(* Logix 5000 project; controller PeerController vendor 1 type 14 code 196 rev 37.11; software revision 37.00 *)

TASK Hot_Backup_15ms (periodic, rate 15 ms, priority 8, watchdog 500 ms) : Hot_Backup
TASK MainTask (continuous, watchdog 500 ms) : MainProgram

MODULES
   Local : vendor 1 type 14 code 196 (5069 0, rev 37.11)
      Primary : vendor 1 type 14 code 196 (Ethernet 192.168.0.177, rev 37.1, $76aec895$ RPI 10 ms)
      FLEX5000_EIP : 5094-AENTR (Ethernet 192.168.0.179, rev 6.1, StandardDataDriven RPI 200 ms)
         FLEX5000_EIP_SLOT1 : vendor 1 type 7 code 1217 (5094 1, rev 2.1, StandardDataDriven RPI 5 ms)
END_MODULES

TYPE Hot_Backup_Event_Log :
STRUCT
   Event_Name : STRING;
   Value : DINT;
   DateTime : DINT[7];   // Controller Date & Time of the Event
END_STRUCT
END_TYPE

TYPE Hot_Backup_EventLog_Triggers :
STRUCT
   Peer_RunMode : BOOL;
   Peer_ProgramMode : BOOL;
   Peer_ConnectionFailed : BOOL;
   Peer_ConnectionOK : BOOL;
   Peer_Owns_Outputs : BOOL;
   Local_Owns_Outputs : BOOL;
   Manual_SwitchOver_Initiated : BOOL;
   Local_Outputs_Inhibited : BOOL;
   Local_Outputs_Uninhibited : BOOL;
   Peer_Ready : BOOL;
   SwitchoverDelayTimerDone : BOOL;
   Peer_ControllerFault : BOOL;
END_STRUCT
END_TYPE

TYPE Hot_Backup_HMI_Interface :
STRUCT
   ClearEventLog : BOOL;
   Switchover : BOOL;
END_STRUCT
END_TYPE

TYPE Hot_Backup_Interface :
STRUCT
   Sts_ConnectionStatus : CONNECTION_STATUS;   // Produced / Consumed connection status
   Sts_ActionDelay : BOOL;   // Set to "1" when the peer action delay timer is timing.
   Sts_Faulted : BOOL;   // Set to "1" when the peer is faulted
   Sts_OutputsOwned : BOOL;   // Set to "1" when the local controller is the owner of the outputs.
   Sts_OutputInhibitRequest : BOOL;   // Set to "1" when the local controller is manually requesting the peer to inhibit its Outputs
   Fbk_OutputInhibitRequest : BOOL;
END_STRUCT
END_TYPE

ADD_ON_INSTRUCTION Hot_Backup   (* revision 2.0, ExecutePrescan *)
// Compact Logix Hot Backup AOI
VAR_INPUT
   Sts_OutputsInhibited : BOOL; {required}
   Sts_OutputsFaulted : BOOL; {required}
   Cfg_PwrUp_Status : BOOL; {visible}
END_VAR
VAR_OUTPUT
   Cmd_InhibitOutputs : BOOL; {access Read Only, visible}
   Cmd_UninhibitOutputs : BOOL; {access Read Only, visible}
   Sts_PeerReady : BOOL; {access Read Only}
   Sts_Primary : BOOL; {access Read Only, visible}
   Sts_Secondary : BOOL; {access Read Only, visible}
   Sts_PostActionDelay : BOOL; {access Read Only}
END_VAR
VAR_IN_OUT
   PEER_Consumed : Hot_Backup_Interface; {required}
   PEER_Produced : Hot_Backup_Interface; {required}
   HMI_Cmd : Hot_Backup_HMI_Interface; {required}
   HMI_HandShake : Hot_Backup_HMI_Interface; {required}
   HMI_Event_Log : Hot_Backup_Event_Log[10]; {required}   // Contains the 5 most recent event log entries for viewing on the HMI.
END_VAR
VAR
   State : DINT; {access None}
   Int_StartUp_Delay : TIMER := (PRE := 10000); {access None}
   Int_PostAction_Delay : TIMER := (PRE := 60000); {access None}
   State_Processed : BOOL; {access None}
   State_1_Transition : BOOL; {access None}
   State_2_Transition : BOOL; {access None}
   State_3_Transition : BOOL; {access None}
   State_4_Transition : BOOL; {access None}
   ONS : DINT; {access None}
   State_5_Transition : BOOL; {access None}
   Cmd_Inhibit_FromPeer : BOOL; {access None}
   Sts_OutputsOwnerless : BOOL; {access None}
   State_6_Transition : BOOL; {access None}
   Event_Log : Hot_Backup_Event_Log[100];
   Event_Log_Entry : Hot_Backup_Event_Log;
   Event_Log_Index : DINT;
   Event_Log_Name_List : STRING[15] := ([0] := 'Peer in Run Mode', [1] := 'Peer in Program Mode', [2] := 'Peer Connection Failed', [3] := 'Local Outputs Inhibited', [4] := 'Peer Connection OK', [5] := 'Switchover Delay Timer Done', [6] := 'Power Up - First Scan Bit Set', [7] := 'Local Outputs Uninhibited', [8] := 'Peer Owns Outputs', [9] := 'Local Owns Outputs', [10] := 'Manual Switchover Initiated', [11] := 'Peer Controller Major Fault', [12] := 'Peer is Ready');   // Listing of the predefined Event Names
   Event_Log_Triggers : Hot_Backup_EventLog_Triggers; {access None}
   First_Scan : BOOL; {access None}
END_VAR

ROUTINE Logic   (* ladder *)
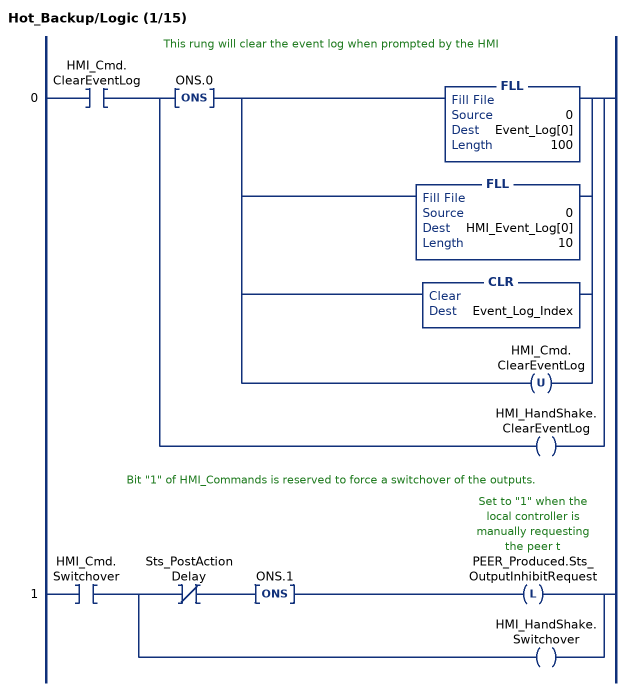
   // This rung will clear the event log when prompted by the HMI
   0: XIC(HMI_Cmd.ClearEventLog)[ONS(ONS.0) [FLL(0,Event_Log[0],100) ,FLL(0,HMI_Event_Log[0],10) ,CLR(Event_Log_Index) ,OTU(HMI_Cmd.ClearEventLog) ] ,OTE(HMI_HandShake.ClearEventLog) ];
   // Bit "1" of HMI_Commands is reserved to force a switchover of the outputs.
   1: XIC(HMI_Cmd.Switchover)[XIO(Sts_PostActionDelay) ONS(ONS.1) OTL(PEER_Produced.Sts_OutputInhibitRequest) ,OTE(HMI_HandShake.Switchover) ];
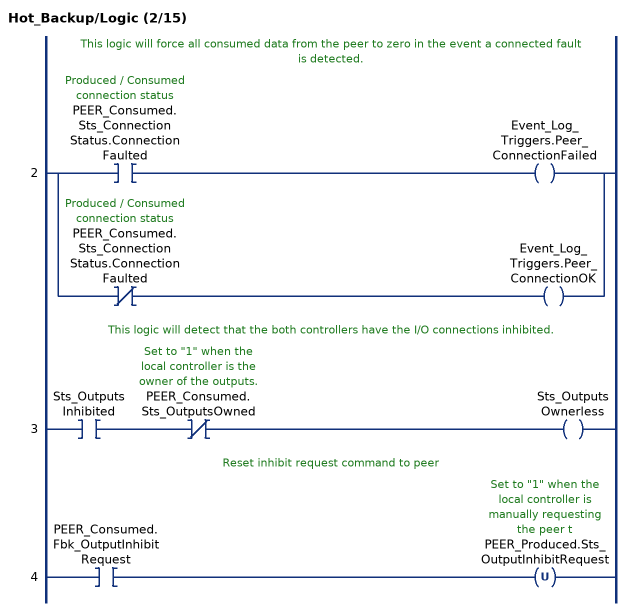
   // This logic will force all consumed data from the peer to zero in the event a connected fault is detected.
   2: [XIC(PEER_Consumed.Sts_ConnectionStatus.ConnectionFaulted) OTE(Event_Log_Triggers.Peer_ConnectionFailed) ,XIO(PEER_Consumed.Sts_ConnectionStatus.ConnectionFaulted) OTE(Event_Log_Triggers.Peer_ConnectionOK) ];
   // This logic will detect that the both controllers have the I/O connections inhibited.
   3: XIC(Sts_OutputsInhibited)XIO(PEER_Consumed.Sts_OutputsOwned)OTE(Sts_OutputsOwnerless);
   // Reset inhibit request command to peer
   4: XIC(PEER_Consumed.Fbk_OutputInhibitRequest)OTU(PEER_Produced.Sts_OutputInhibitRequest);
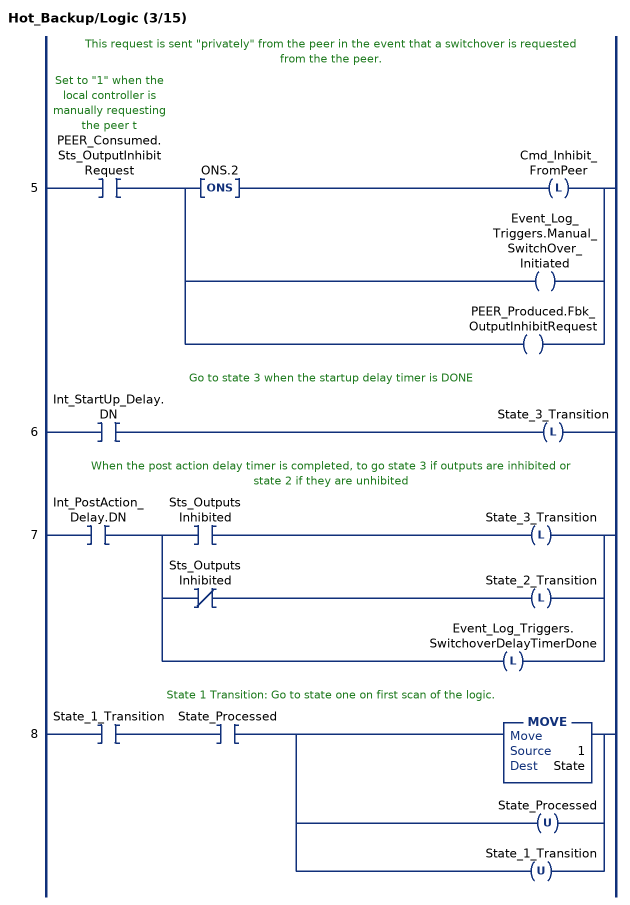
   // This request is sent "privately" from the peer in the event that a switchover is requested from the the peer.
   5: XIC(PEER_Consumed.Sts_OutputInhibitRequest)[ONS(ONS.2) OTL(Cmd_Inhibit_FromPeer) ,OTE(Event_Log_Triggers.Manual_SwitchOver_Initiated) ,OTE(PEER_Produced.Fbk_OutputInhibitRequest) ];
   // Go to state 3 when the startup delay timer is DONE
   6: XIC(Int_StartUp_Delay.DN)OTL(State_3_Transition);
   // When the post action delay timer is completed, to go state 3 if outputs are inhibited or state 2 if they are unhibited
   7: XIC(Int_PostAction_Delay.DN)[XIC(Sts_OutputsInhibited) OTL(State_3_Transition) ,XIO(Sts_OutputsInhibited) OTL(State_2_Transition) ,OTL(Event_Log_Triggers.SwitchoverDelayTimerDone) ];
   // State 1 Transition: Go to state one on first scan of the logic.
   8: XIC(State_1_Transition)XIC(State_Processed)[MOVE(1,State) ,OTU(State_Processed) ,OTU(State_1_Transition) ];
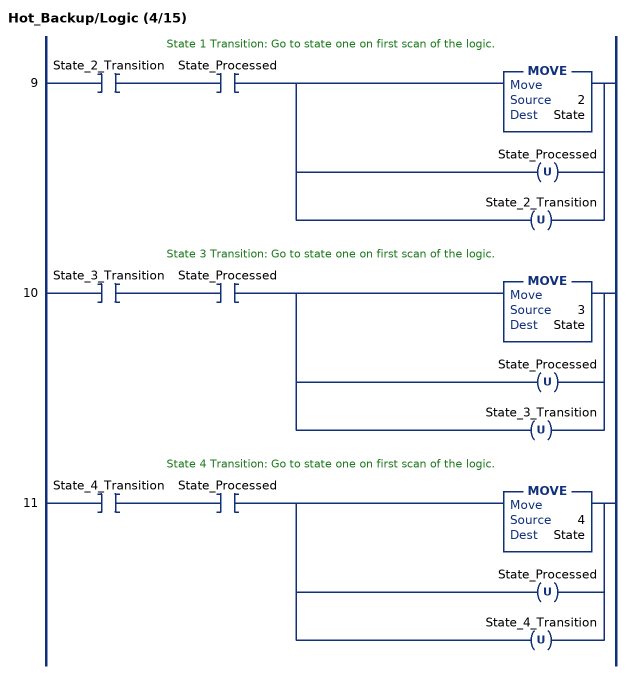
   // State 1 Transition: Go to state one on first scan of the logic.
   9: XIC(State_2_Transition)XIC(State_Processed)[MOVE(2,State) ,OTU(State_Processed) ,OTU(State_2_Transition) ];
   // State 3 Transition: Go to state one on first scan of the logic.
   10: XIC(State_3_Transition)XIC(State_Processed)[MOVE(3,State) ,OTU(State_Processed) ,OTU(State_3_Transition) ];
   // State 4 Transition: Go to state one on first scan of the logic.
   11: XIC(State_4_Transition)XIC(State_Processed)[MOVE(4,State) ,OTU(State_Processed) ,OTU(State_4_Transition) ];
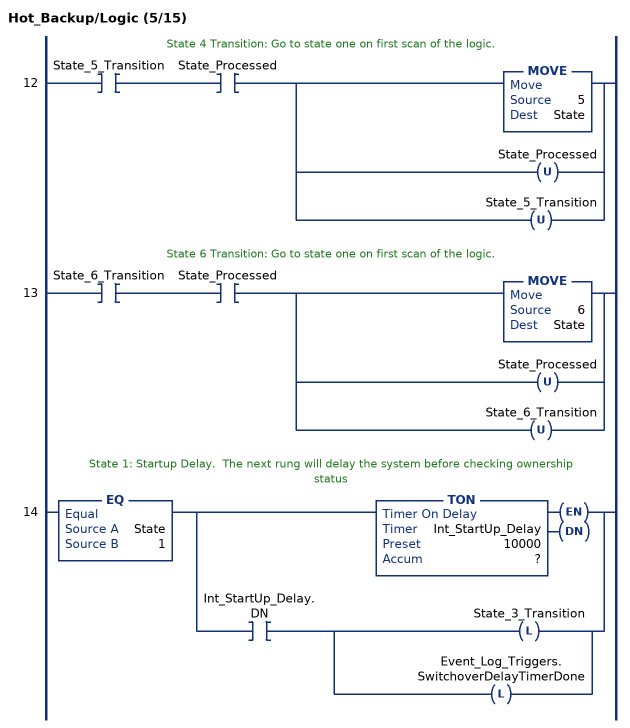
   // State 4 Transition: Go to state one on first scan of the logic.
   12: XIC(State_5_Transition)XIC(State_Processed)[MOVE(5,State) ,OTU(State_Processed) ,OTU(State_5_Transition) ];
   // State 6 Transition: Go to state one on first scan of the logic.
   13: XIC(State_6_Transition)XIC(State_Processed)[MOVE(6,State) ,OTU(State_Processed) ,OTU(State_6_Transition) ];
   // State 1: Startup Delay.  The next rung will delay the system before checking ownership status
   14: EQ(State,1)[TON(Int_StartUp_Delay,?,?) ,XIC(Int_StartUp_Delay.DN) [OTL(State_3_Transition) ,OTL(Event_Log_Triggers.SwitchoverDelayTimerDone) ] ];
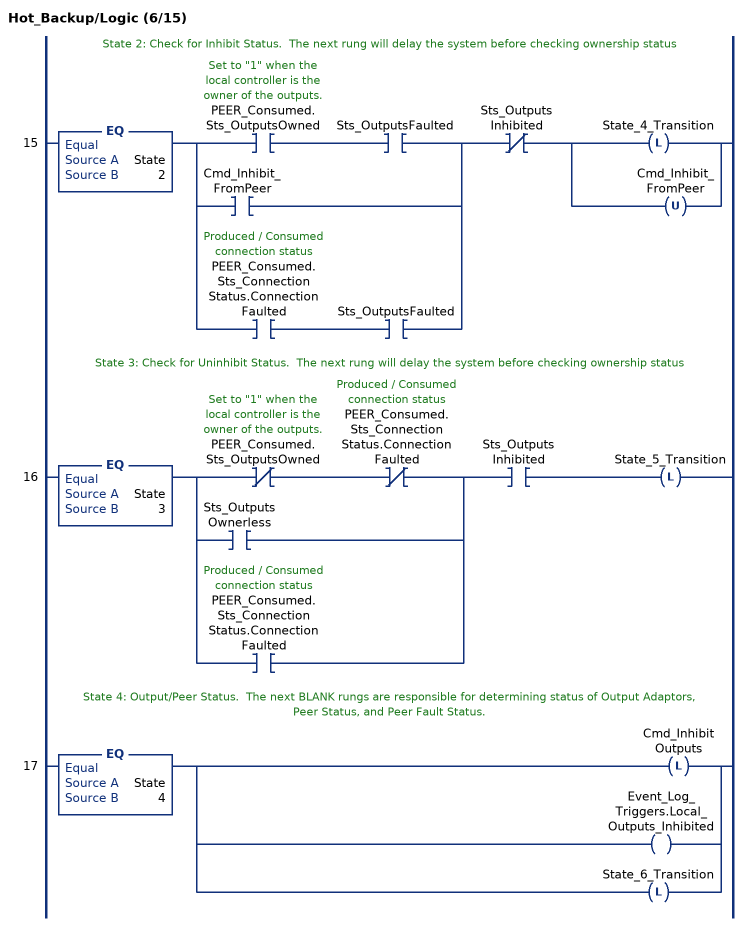
   // State 2: Check for Inhibit Status.  The next rung will delay the system before checking ownership status
   15: EQ(State,2)[XIC(PEER_Consumed.Sts_OutputsOwned) XIC(Sts_OutputsFaulted) ,XIC(Cmd_Inhibit_FromPeer) ,XIC(PEER_Consumed.Sts_ConnectionStatus.ConnectionFaulted) XIC(Sts_OutputsFaulted) ]XIO(Sts_OutputsInhibited)[OTL(State_4_Transition) ,OTU(Cmd_Inhibit_FromPeer) ];
   // State 3: Check for Uninhibit Status.  The next rung will delay the system before checking ownership status
   16: EQ(State,3)[XIO(PEER_Consumed.Sts_OutputsOwned) XIO(PEER_Consumed.Sts_ConnectionStatus.ConnectionFaulted) ,XIC(Sts_OutputsOwnerless) ,XIC(PEER_Consumed.Sts_ConnectionStatus.ConnectionFaulted) ]XIC(Sts_OutputsInhibited)OTL(State_5_Transition);
   // State 4: Output/Peer Status.  The next BLANK rungs are responsible for determining status of Output Adaptors, Peer Status, and Peer Fault Status.
   17: EQ(State,4)[OTL(Cmd_InhibitOutputs) ,OTE(Event_Log_Triggers.Local_Outputs_Inhibited) ,OTL(State_6_Transition) ];
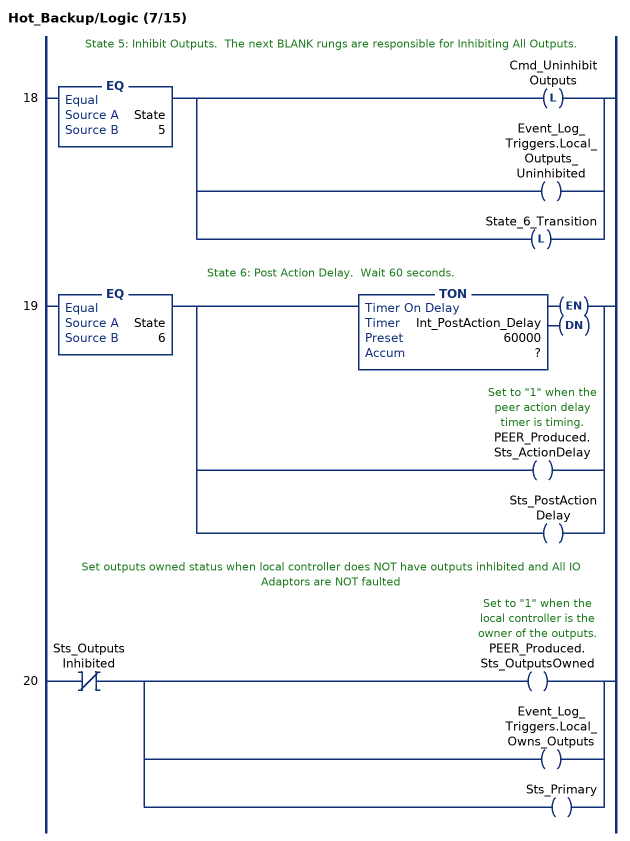
   // State 5: Inhibit Outputs.  The next BLANK rungs are responsible for Inhibiting All Outputs.
   18: EQ(State,5)[OTL(Cmd_UninhibitOutputs) ,OTE(Event_Log_Triggers.Local_Outputs_Uninhibited) ,OTL(State_6_Transition) ];
   // State 6: Post Action Delay.  Wait 60 seconds.
   19: EQ(State,6)[TON(Int_PostAction_Delay,?,?) ,OTE(PEER_Produced.Sts_ActionDelay) ,OTE(Sts_PostActionDelay) ];
   // Set outputs owned status when local controller does NOT have outputs inhibited and All IO Adaptors are NOT faulted
   20: XIO(Sts_OutputsInhibited)[OTE(PEER_Produced.Sts_OutputsOwned) ,OTE(Event_Log_Triggers.Local_Owns_Outputs) ,OTE(Sts_Primary) ];
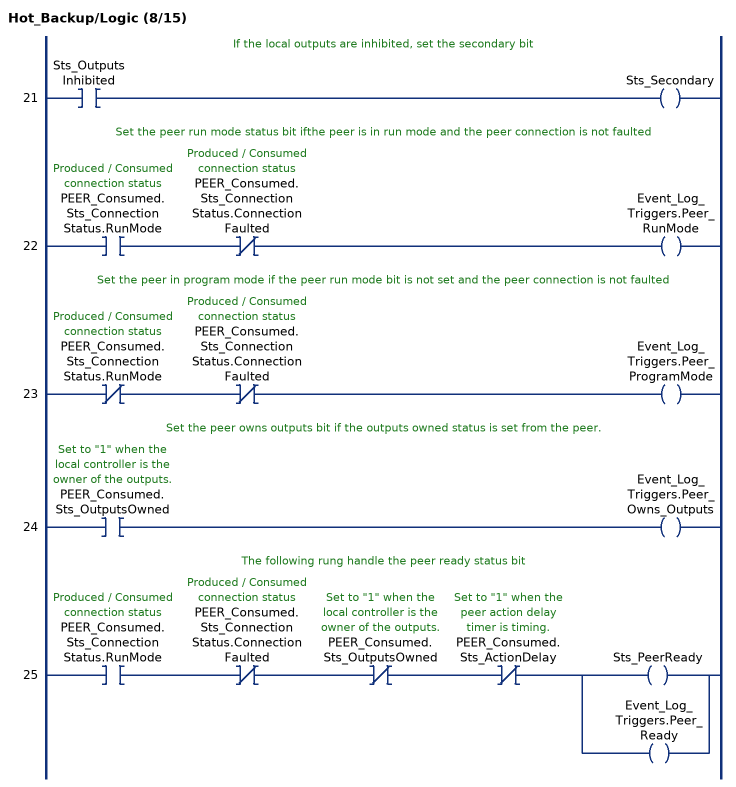
   // If the local outputs are inhibited, set the secondary bit
   21: XIC(Sts_OutputsInhibited)OTE(Sts_Secondary);
   // Set the peer run mode status bit ifthe peer is in run mode and the peer connection is not faulted
   22: XIC(PEER_Consumed.Sts_ConnectionStatus.RunMode)XIO(PEER_Consumed.Sts_ConnectionStatus.ConnectionFaulted)OTE(Event_Log_Triggers.Peer_RunMode);
   // Set the peer in program mode if the peer run mode bit is not set and the peer connection is not faulted
   23: XIO(PEER_Consumed.Sts_ConnectionStatus.RunMode)XIO(PEER_Consumed.Sts_ConnectionStatus.ConnectionFaulted)OTE(Event_Log_Triggers.Peer_ProgramMode);
   // Set the peer owns outputs bit if the outputs owned status is set from the peer.
   24: XIC(PEER_Consumed.Sts_OutputsOwned)OTE(Event_Log_Triggers.Peer_Owns_Outputs);
   // The following rung handle the peer ready status bit
   25: XIC(PEER_Consumed.Sts_ConnectionStatus.RunMode)XIO(PEER_Consumed.Sts_ConnectionStatus.ConnectionFaulted)XIO(PEER_Consumed.Sts_OutputsOwned)XIO(PEER_Consumed.Sts_ActionDelay)[OTE(Sts_PeerReady) ,OTE(Event_Log_Triggers.Peer_Ready) ];
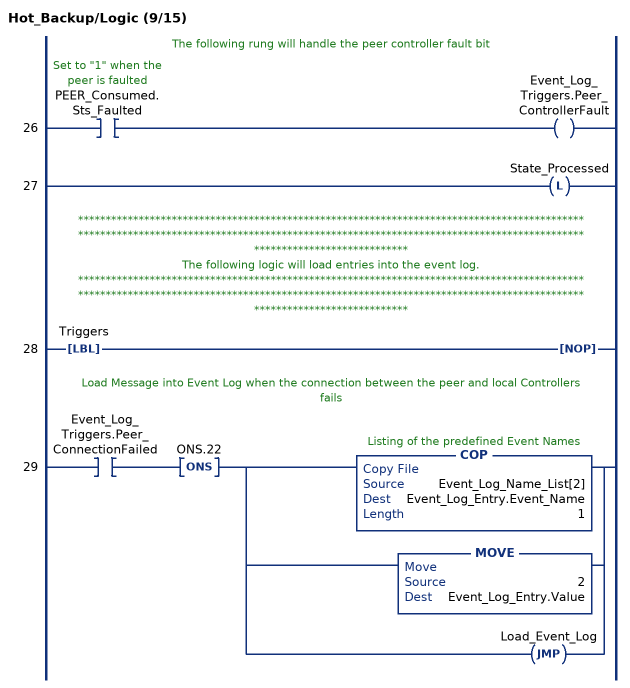
   // The following rung will handle the peer controller fault bit
   26: XIC(PEER_Consumed.Sts_Faulted)OTE(Event_Log_Triggers.Peer_ControllerFault);
   27: OTL(State_Processed);
   // ********************************************************************************************************************************************************************************************************************
   // The following logic will load entries into the event log.
   // ********************************************************************************************************************************************************************************************************************
   28: LBL(Triggers)NOP();
   // Load Message into Event Log when the connection between the peer and local Controllers fails
   29: XIC(Event_Log_Triggers.Peer_ConnectionFailed)ONS(ONS.22)[COP(Event_Log_Name_List[2],Event_Log_Entry.Event_Name,1) ,MOVE(2,Event_Log_Entry.Value) ,JMP(Load_Event_Log) ];
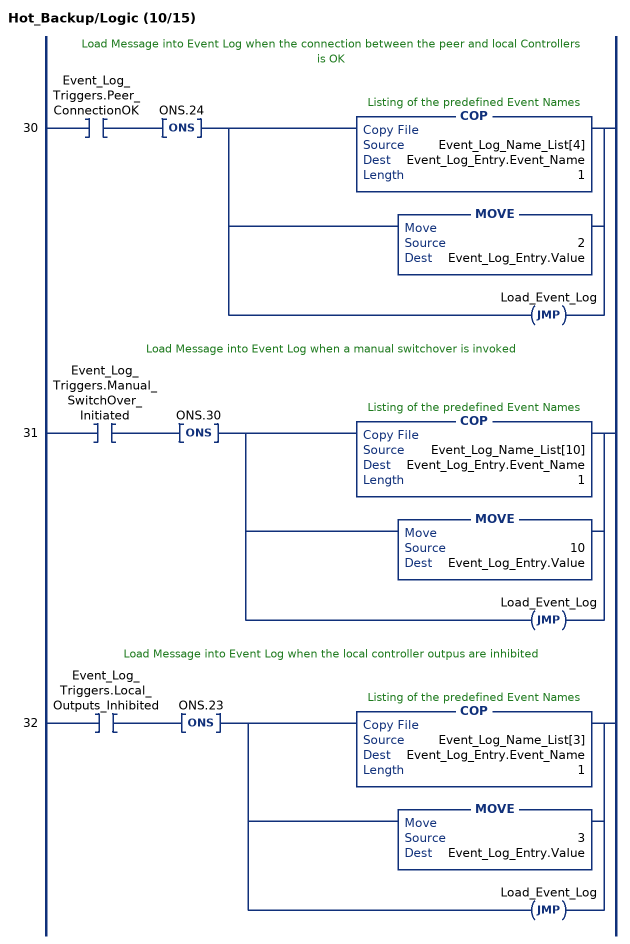
   // Load Message into Event Log when the connection between the peer and local Controllers is OK
   30: XIC(Event_Log_Triggers.Peer_ConnectionOK)ONS(ONS.24)[COP(Event_Log_Name_List[4],Event_Log_Entry.Event_Name,1) ,MOVE(2,Event_Log_Entry.Value) ,JMP(Load_Event_Log) ];
   // Load Message into Event Log when a manual switchover is invoked
   31: XIC(Event_Log_Triggers.Manual_SwitchOver_Initiated)ONS(ONS.30)[COP(Event_Log_Name_List[10],Event_Log_Entry.Event_Name,1) ,MOVE(10,Event_Log_Entry.Value) ,JMP(Load_Event_Log) ];
   // Load Message into Event Log when the local controller outpus are inhibited
   32: XIC(Event_Log_Triggers.Local_Outputs_Inhibited)ONS(ONS.23)[COP(Event_Log_Name_List[3],Event_Log_Entry.Event_Name,1) ,MOVE(3,Event_Log_Entry.Value) ,JMP(Load_Event_Log) ];
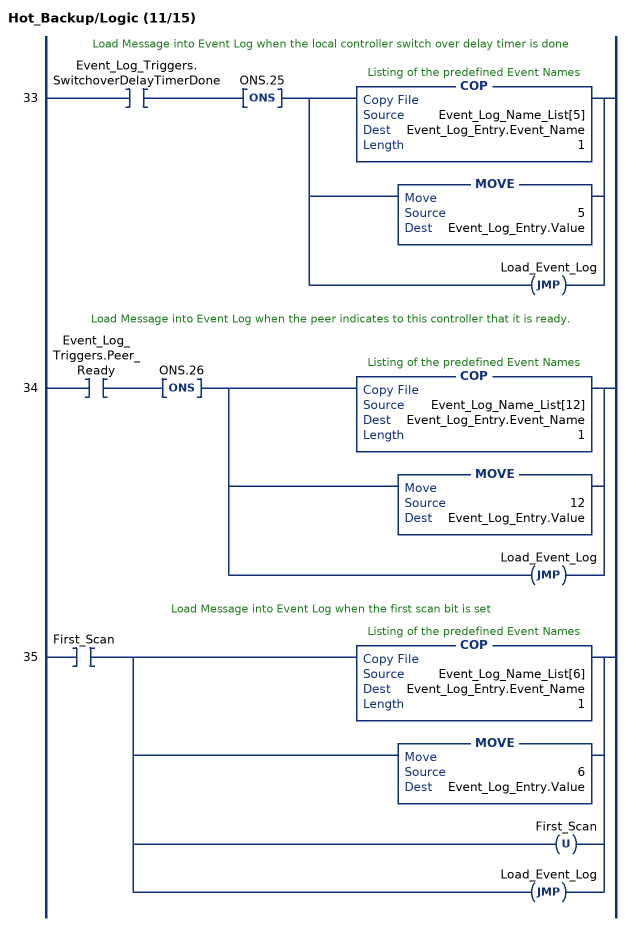
   // Load Message into Event Log when the local controller switch over delay timer is done
   33: XIC(Event_Log_Triggers.SwitchoverDelayTimerDone)ONS(ONS.25)[COP(Event_Log_Name_List[5],Event_Log_Entry.Event_Name,1) ,MOVE(5,Event_Log_Entry.Value) ,JMP(Load_Event_Log) ];
   // Load Message into Event Log when the peer indicates to this controller that it is ready.
   34: XIC(Event_Log_Triggers.Peer_Ready)ONS(ONS.26)[COP(Event_Log_Name_List[12],Event_Log_Entry.Event_Name,1) ,MOVE(12,Event_Log_Entry.Value) ,JMP(Load_Event_Log) ];
   // Load Message into Event Log when the first scan bit is set
   35: XIC(First_Scan)[COP(Event_Log_Name_List[6],Event_Log_Entry.Event_Name,1) ,MOVE(6,Event_Log_Entry.Value) ,OTU(First_Scan) ,JMP(Load_Event_Log) ];
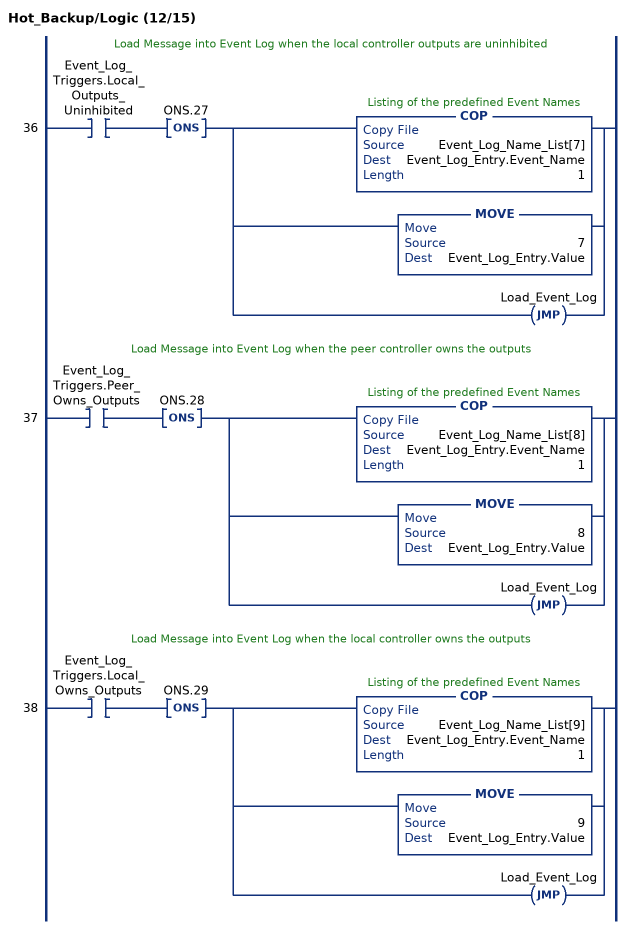
   // Load Message into Event Log when the local controller outputs are uninhibited
   36: XIC(Event_Log_Triggers.Local_Outputs_Uninhibited)ONS(ONS.27)[COP(Event_Log_Name_List[7],Event_Log_Entry.Event_Name,1) ,MOVE(7,Event_Log_Entry.Value) ,JMP(Load_Event_Log) ];
   // Load Message into Event Log when the peer controller owns the outputs
   37: XIC(Event_Log_Triggers.Peer_Owns_Outputs)ONS(ONS.28)[COP(Event_Log_Name_List[8],Event_Log_Entry.Event_Name,1) ,MOVE(8,Event_Log_Entry.Value) ,JMP(Load_Event_Log) ];
   // Load Message into Event Log when the local controller owns the outputs
   38: XIC(Event_Log_Triggers.Local_Owns_Outputs)ONS(ONS.29)[COP(Event_Log_Name_List[9],Event_Log_Entry.Event_Name,1) ,MOVE(9,Event_Log_Entry.Value) ,JMP(Load_Event_Log) ];
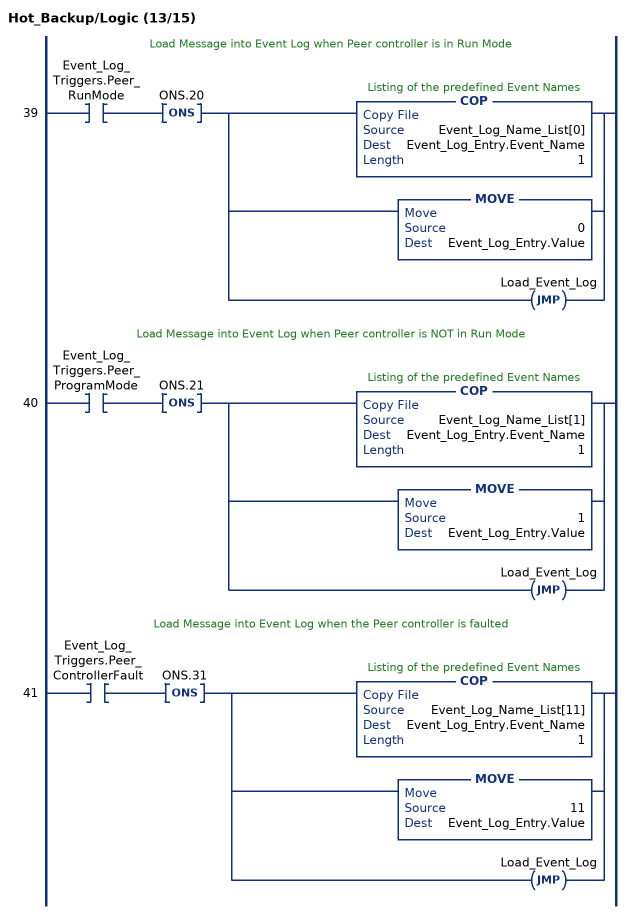
   // Load Message into Event Log when Peer controller is in Run Mode
   39: XIC(Event_Log_Triggers.Peer_RunMode)ONS(ONS.20)[COP(Event_Log_Name_List[0],Event_Log_Entry.Event_Name,1) ,MOVE(0,Event_Log_Entry.Value) ,JMP(Load_Event_Log) ];
   // Load Message into Event Log when Peer controller is NOT in Run Mode
   40: XIC(Event_Log_Triggers.Peer_ProgramMode)ONS(ONS.21)[COP(Event_Log_Name_List[1],Event_Log_Entry.Event_Name,1) ,MOVE(1,Event_Log_Entry.Value) ,JMP(Load_Event_Log) ];
   // Load Message into Event Log when the Peer controller is faulted
   41: XIC(Event_Log_Triggers.Peer_ControllerFault)ONS(ONS.31)[COP(Event_Log_Name_List[11],Event_Log_Entry.Event_Name,1) ,MOVE(11,Event_Log_Entry.Value) ,JMP(Load_Event_Log) ];
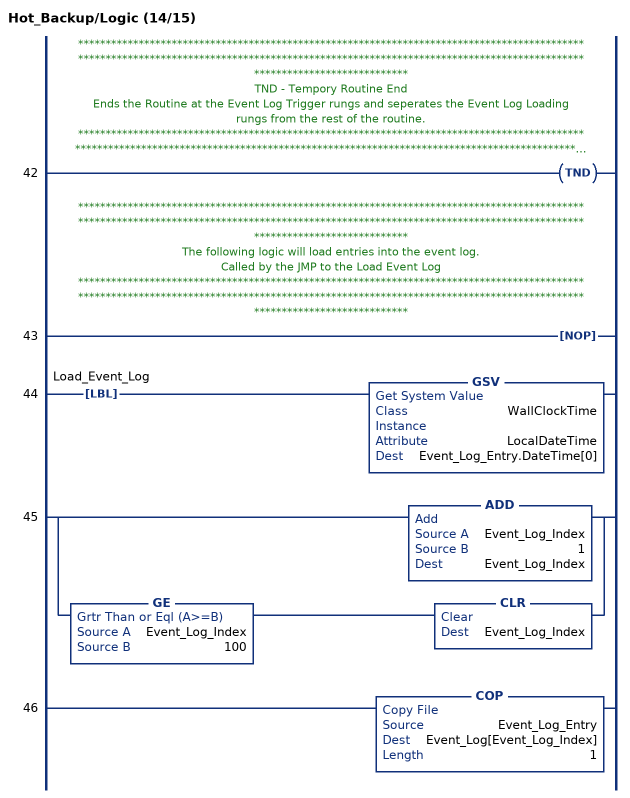
   // ********************************************************************************************************************************************************************************************************************
   // TND - Tempory Routine End
   // Ends the Routine at the Event Log Trigger rungs and seperates the Event Log Loading rungs from the rest of the routine.
   // ********************************************************************************************************************************************************************************************************************
   42: TND();
   // ********************************************************************************************************************************************************************************************************************
   // The following logic will load entries into the event log.
   // Called by the JMP to the Load Event Log
   // ********************************************************************************************************************************************************************************************************************
   43: NOP();
   44: LBL(Load_Event_Log)GSV(WallClockTime,,LocalDateTime,Event_Log_Entry.DateTime[0]);
   45: [ADD(Event_Log_Index,1,Event_Log_Index) ,GE(Event_Log_Index,100) CLR(Event_Log_Index) ];
   46: COP(Event_Log_Entry,Event_Log[Event_Log_Index],1);
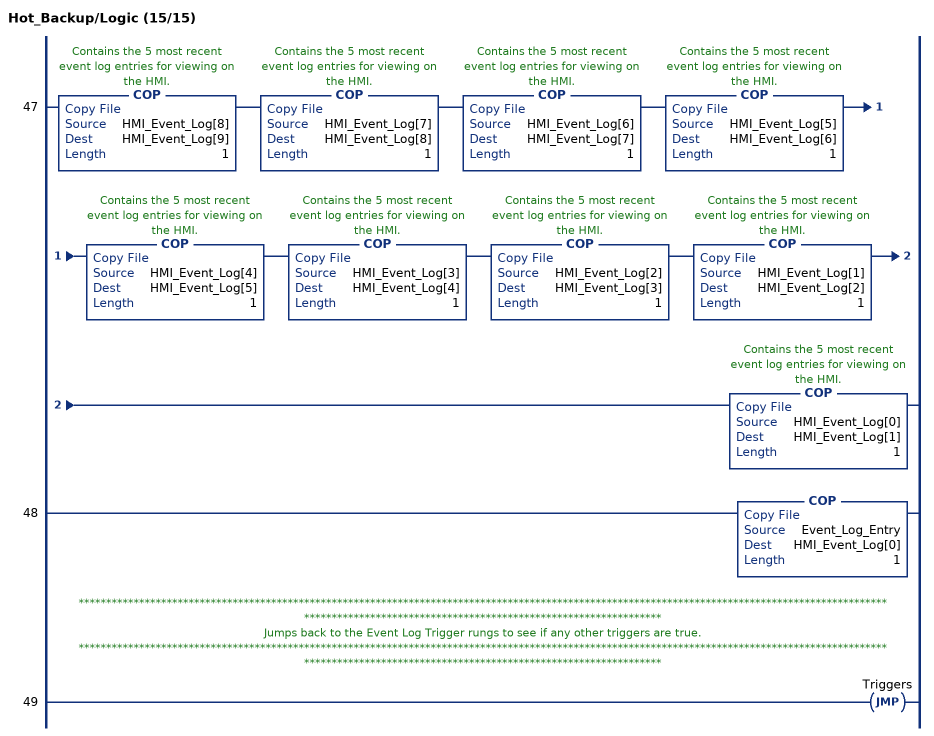
   47: COP(HMI_Event_Log[8],HMI_Event_Log[9],1)COP(HMI_Event_Log[7],HMI_Event_Log[8],1)COP(HMI_Event_Log[6],HMI_Event_Log[7],1)COP(HMI_Event_Log[5],HMI_Event_Log[6],1)COP(HMI_Event_Log[4],HMI_Event_Log[5],1)COP(HMI_Event_Log[3],HMI_Event_Log[4],1)COP(HMI_Event_Log[2],HMI_Event_Log[3],1)COP(HMI_Event_Log[1],HMI_Event_Log[2],1)COP(HMI_Event_Log[0],HMI_Event_Log[1],1);
   48: COP(Event_Log_Entry,HMI_Event_Log[0],1);
   // ********************************************************************************************************************************************************************************************************************
   // Jumps back to the Event Log Trigger rungs to see if any other triggers are true.
   // ********************************************************************************************************************************************************************************************************************
   49: JMP(Triggers);
END_ROUTINE

ROUTINE Prescan   (* ladder *)
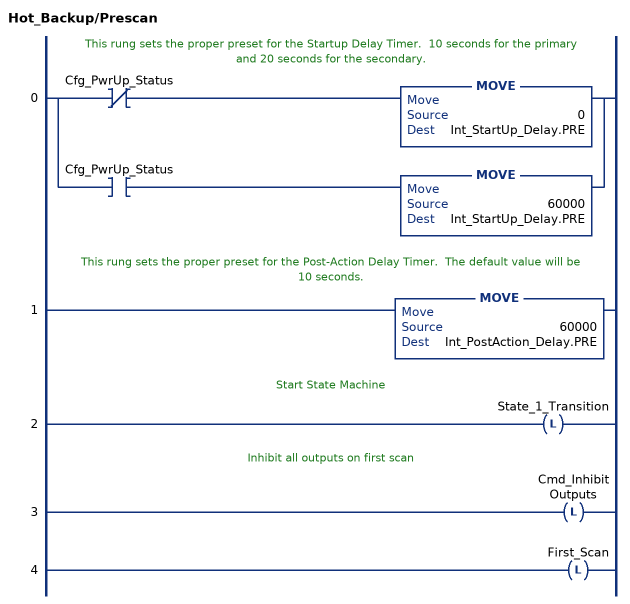
   // This rung sets the proper preset for the Startup Delay Timer.  10 seconds for the primary and 20 seconds for the secondary.
   0: [XIO(Cfg_PwrUp_Status) MOVE(0,Int_StartUp_Delay.PRE) ,XIC(Cfg_PwrUp_Status) MOVE(60000,Int_StartUp_Delay.PRE) ];
   // This rung sets the proper preset for the Post-Action Delay Timer.  The default value will be 10 seconds.
   1: MOVE(60000,Int_PostAction_Delay.PRE);
   // Start State Machine
   2: OTL(State_1_Transition);
   // Inhibit all outputs on first scan
   3: OTL(Cmd_InhibitOutputs);
   4: OTL(First_Scan);
END_ROUTINE
END_ADD_ON_INSTRUCTION

VAR_GLOBAL   (* controller tags *)
   Array : DINT[10];
   DINT : DINT;
   HMI_Cmd : Hot_Backup_HMI_Interface;
   HMI_Event_Log : Hot_Backup_Event_Log[10];
   HMI_Handshake : Hot_Backup_HMI_Interface;
   Manual_Switchover_PB : BOOL;
   PEER_HB_Consume : Hot_Backup_Interface := (Sts_ConnectionStatus.RunMode := 1, Sts_OutputsOwned := 1);   // Consumed data from the parter controller
   PEER_HB_Produce : Hot_Backup_Interface := (Sts_ConnectionStatus.RunMode := 1, Sts_OutputsOwned := 1); {produced}   // Produced data to the peer controller.
   REAL : REAL;
END_VAR

PROGRAM Fault_Program   (* main routine Fault_Main *)
VAR
   Val_ModuleMode : DINT;
END_VAR

ROUTINE Fault_Main   (* ladder *)
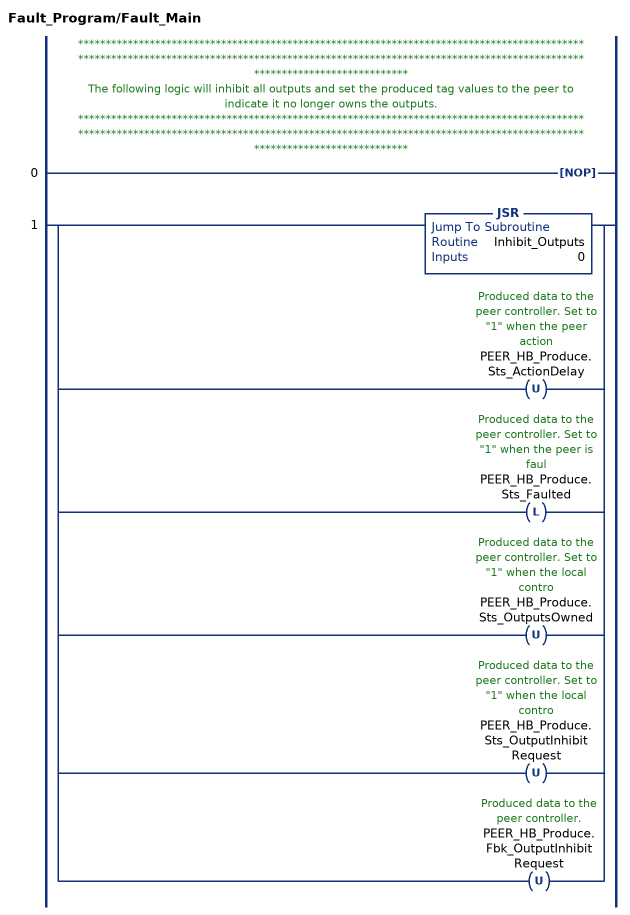
   // ********************************************************************************************************************************************************************************************************************
   // The following logic will inhibit all outputs and set the produced tag values to the peer to indicate it no longer owns the outputs.
   // ********************************************************************************************************************************************************************************************************************
   0: NOP();
   1: [JSR(Inhibit_Outputs,0) ,OTU(PEER_HB_Produce.Sts_ActionDelay) ,OTL(PEER_HB_Produce.Sts_Faulted) ,OTU(PEER_HB_Produce.Sts_OutputsOwned) ,OTU(PEER_HB_Produce.Sts_OutputInhibitRequest) ,OTU(PEER_HB_Produce.Fbk_OutputInhibitRequest) ];
END_ROUTINE

ROUTINE Inhibit_Outputs   (* ladder *)
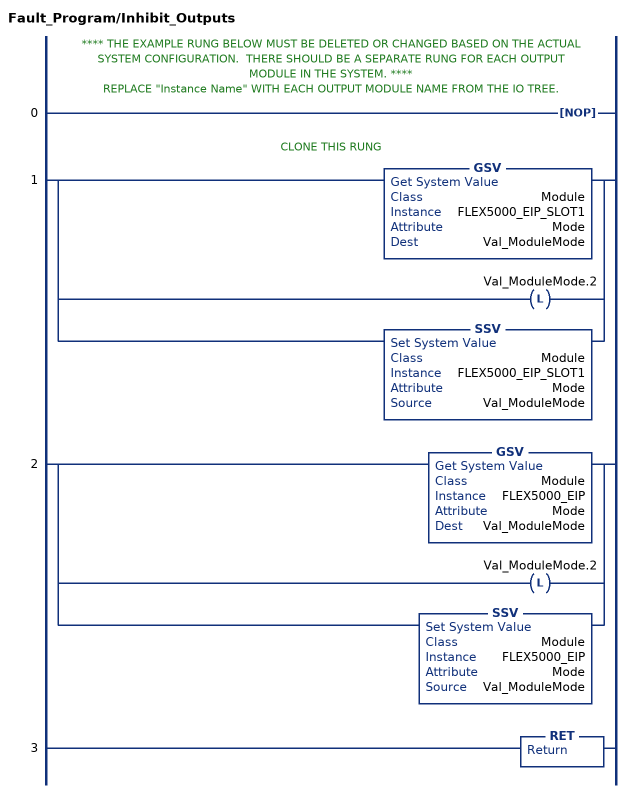
   // **** THE EXAMPLE RUNG BELOW MUST BE DELETED OR CHANGED BASED ON THE ACTUAL SYSTEM CONFIGURATION.  THERE SHOULD BE A SEPARATE RUNG FOR EACH OUTPUT MODULE IN THE SYSTEM. ****
   // REPLACE "Instance Name" WITH EACH OUTPUT MODULE NAME FROM THE IO TREE.
   0: NOP();
   // CLONE THIS RUNG
   1: [GSV(Module,FLEX5000_EIP_SLOT1,Mode,Val_ModuleMode) ,OTL(Val_ModuleMode.2) ,SSV(Module,FLEX5000_EIP_SLOT1,Mode,Val_ModuleMode) ];
   2: [GSV(Module,FLEX5000_EIP,Mode,Val_ModuleMode) ,OTL(Val_ModuleMode.2) ,SSV(Module,FLEX5000_EIP,Mode,Val_ModuleMode) ];
   3: RET();
END_ROUTINE
END_PROGRAM
